ABB RobotStudio station: EstaciónDibujo_20220828-163813.rsstn

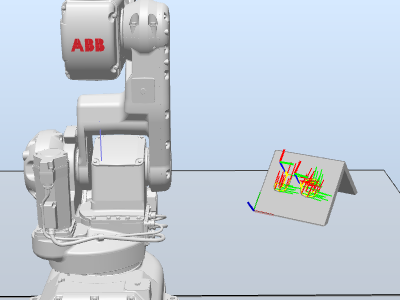
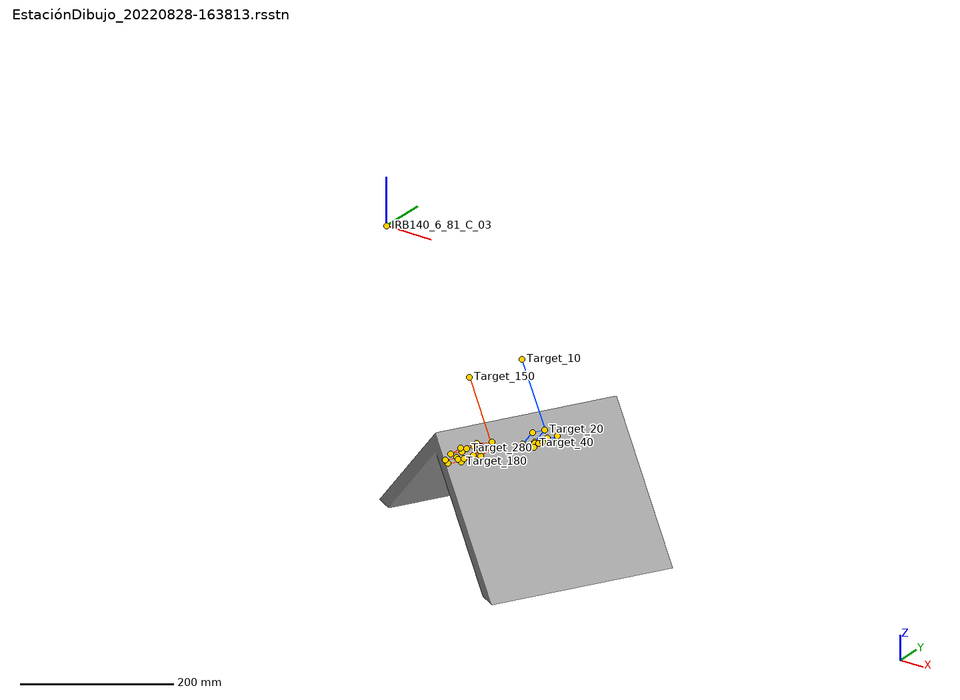
[picture v1: parts stored in the station drawn from their meshes, with robot base, taught points and paths (robot models come from the ABB library and are not in the file)]
Station EstaciónDibujo (saved by RobotStudio 22.2.9947.0)
Controller ControladorDibujo
  mechanical unit ROB_1: IRB140_6_81_C_03, 6 joints, base frame (0, 0, 0) mm
Layout (positions relative to the parent item):
  - IRB140_6_81_C_03 [mechanism, from Robots\IRB140_6_81_C_G_03.rslib] at (0, 0, 0) mm; joint values [0, 0, 0, 0, 0, 0] (rad or m)
  - Tablero [part] at (588.81, -446.49, 0) mm, rotated rx 90 ry 0 rz -120 deg, size 260 x 173.2 x 346.5 mm
  - HerramientaMarcador [mechanism] at (515, 0, 712) mm, rotated rx 0 ry 90 rz 0 deg
      TCP PuntaMarcador at (58.47, 0, 120.68) mm, rotated rx 0 ry 40 rz 0 deg
      links: HerramientaM-Marcador
  - Part_1 [part] at (588.81, -446.49, 0) mm, rotated rx 90 ry 0 rz -120 deg, size 260 x 173.2 x 173.2 mm
Attachment: HerramientaMarcador is attached to IRB140_6_81_C_03 / Link6
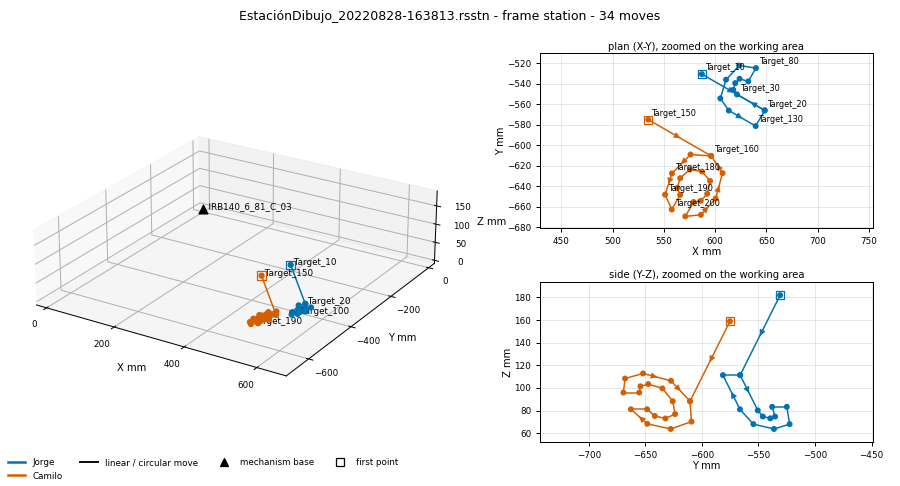
[picture p0: tool path of EstaciónDibujo_20220828-163813.rsstn in frame station, 34 of 36 moves have a stored position in this frame; points joined in program order, loops and branches not executed]
Targets, tools, work objects and paths stored in the station, written as RAPID:
! task T_ROB1
MODULE Module1
  CONST robtarget Target_10:=[[73.955465637,157.243972961,100.000985962],[-0.000003962,0.707387962,0.706825489,0.000002607],[0,0,0,0],[9E+09,9E+09,9E+09,9E+09,9E+09,9E+09]];
  CONST robtarget Target_20:=[[73.955274379,157.244902053,0.000985967],[-0.000003962,0.707387962,0.706825489,0.000002607],[0,0,0,0],[9E+09,9E+09,9E+09,9E+09,9E+09,9E+09]];
  CONST robtarget Target_30:=[[73.920195161,113.145486504,0.000576311],[-0.000003962,0.707387962,0.706825489,0.000002607],[0,0,0,0],[9E+09,9E+09,9E+09,9E+09,9E+09,9E+09]];
  CONST robtarget Target_40:=[[71.888872615,105.530963007,0.00050945],[-0.000003962,0.707387962,0.706825489,0.000002607],[0,0,0,0],[9E+09,9E+09,9E+09,9E+09,9E+09,9E+09]];
  CONST robtarget Target_50:=[[65.240745034,103.225737132,0.000500747],[-0.000003962,0.707387962,0.706825489,0.000002607],[0,0,0,0],[9E+09,9E+09,9E+09,9E+09,9E+09,9E+09]];
  CONST robtarget Target_60:=[[59.480450131,105.398209048,0.000531949],[-0.000003962,0.707387962,0.706825489,0.000002607],[0,0,0,0],[9E+09,9E+09,9E+09,9E+09,9E+09,9E+09]];
  CONST robtarget Target_70:=[[57.436372502,117.608477845,0.000649303],[-0.000003962,0.707387962,0.706825489,0.000002607],[0,0,0,0],[9E+09,9E+09,9E+09,9E+09,9E+09,9E+09]];
  CONST robtarget Target_80:=[[42.489351966,117.620367567,0.000678],[-0.000003962,0.707387962,0.706825489,0.000002607],[0,0,0,0],[9E+09,9E+09,9E+09,9E+09,9E+09,9E+09]];
  CONST robtarget Target_90:=[[48.405321169,95.993812933,0.000465755],[-0.000003962,0.707387962,0.706825489,0.000002607],[0,0,0,0],[9E+09,9E+09,9E+09,9E+09,9E+09,9E+09]];
  CONST robtarget Target_100:=[[66.827562858,89.931887143,0.0003742],[-0.000003962,0.707387962,0.706825489,0.000002607],[0,0,0,0],[9E+09,9E+09,9E+09,9E+09,9E+09,9E+09]];
  CONST robtarget Target_110:=[[85.430597019,95.992885761,0.000394933],[-0.000003962,0.707387962,0.706825489,0.000002607],[0,0,0,0],[9E+09,9E+09,9E+09,9E+09,9E+09,9E+09]];
  CONST robtarget Target_120:=[[91.549595196,114.443606918,0.000554654],[-0.000003962,0.707387962,0.706825489,0.000002607],[0,0,0,0],[9E+09,9E+09,9E+09,9E+09,9E+09,9E+09]];
  CONST robtarget Target_130:=[[91.583630659,157.230879442,0.000952121],[-0.000003962,0.707387962,0.706825489,0.000002607],[0,0,0,0],[9E+09,9E+09,9E+09,9E+09,9E+09,9E+09]];
  CONST robtarget Target_140:=[[73.955274379,157.244902053,0.000985967],[-0.000003962,0.707387962,0.706825489,0.000002607],[0,0,0,0],[9E+09,9E+09,9E+09,9E+09,9E+09,9E+09]];
  CONST jointtarget Home:=[[0,0,0,0,0,0],[9E+09,9E+09,9E+09,9E+09,9E+09,9E+09]];
  CONST robtarget Target_150:=[[138.452714894,124.560220972,100.000558944],[0.000004101,0.745570763,0.666426468,0.000002383],[0,0,0,0],[9E+09,9E+09,9E+09,9E+09,9E+09,9E+09]];
  CONST robtarget Target_160:=[[138.452523635,124.561150062,0.000558949],[0.000004101,0.745570763,0.666426468,0.000002383],[0,0,0,0],[9E+09,9E+09,9E+09,9E+09,9E+09,9E+09]];
  CONST robtarget Target_170:=[[147.331968493,99.024331413,0.000304705],[0.000004101,0.745570763,0.666426468,0.000002383],[0,0,0,0],[9E+09,9E+09,9E+09,9E+09,9E+09,9E+09]];
  CONST robtarget Target_180:=[[172.255402363,89.848023763,0.00017178],[0.000004101,0.745570763,0.666426468,0.000002383],[0,0,0,0],[9E+09,9E+09,9E+09,9E+09,9E+09,9E+09]];
  CONST robtarget Target_190:=[[193.568592092,96.27768983,0.000190755],[0.000004101,0.745570763,0.666426468,0.000002383],[0,0,0,0],[9E+09,9E+09,9E+09,9E+09,9E+09,9E+09]];
  CONST robtarget Target_200:=[[202.91069392,114.469123347,0.000341902],[0.000004101,0.745570763,0.666426468,0.000002383],[0,0,0,0],[9E+09,9E+09,9E+09,9E+09,9E+09,9E+09]];
  CONST robtarget Target_210:=[[186.423331573,114.482238345,0.000373558],[0.000004101,0.745570763,0.666426468,0.000002383],[0,0,0,0],[9E+09,9E+09,9E+09,9E+09,9E+09,9E+09]];
  CONST robtarget Target_220:=[[181.881209734,106.099540689,0.000304363],[0.000004101,0.745570763,0.666426468,0.000002383],[0,0,0,0],[9E+09,9E+09,9E+09,9E+09,9E+09,9E+09]];
  CONST robtarget Target_230:=[[172.322889602,102.969408624,0.000293562],[0.000004101,0.745570763,0.666426468,0.000002383],[0,0,0,0],[9E+09,9E+09,9E+09,9E+09,9E+09,9E+09]];
  CONST robtarget Target_240:=[[160.26125798,108.484302356,0.000367869],[0.000004101,0.745570763,0.666426468,0.000002383],[0,0,0,0],[9E+09,9E+09,9E+09,9E+09,9E+09,9E+09]];
  CONST robtarget Target_250:=[[156.080834535,124.490077756,0.000524572],[0.000004101,0.745570763,0.666426468,0.000002383],[0,0,0,0],[9E+09,9E+09,9E+09,9E+09,9E+09,9E+09]];
  CONST robtarget Target_260:=[[160.144183026,140.60339505,0.000666508],[0.000004101,0.745570763,0.666426468,0.000002383],[0,0,0,0],[9E+09,9E+09,9E+09,9E+09,9E+09,9E+09]];
  CONST robtarget Target_270:=[[172.357106589,145.984879936,0.000693148],[0.000004673,-0.031268643,0.999511016,0.000000809],[0,0,0,0],[9E+09,9E+09,9E+09,9E+09,9E+09,9E+09]];
  CONST robtarget Target_280:=[[181.48283441,143.182183899,0.000649655],[0.000004673,-0.031268643,0.999511016,0.000000809],[0,0,0,0],[9E+09,9E+09,9E+09,9E+09,9E+09,9E+09]];
  CONST robtarget Target_290:=[[185.926493609,135.362835763,0.000568508],[0.000004585,0.055963469,0.998432817,0.000001213],[0,0,0,0],[9E+09,9E+09,9E+09,9E+09,9E+09,9E+09]];
  CONST robtarget Target_300:=[[202.071557775,135.349993048,0.00053751],[0.000004673,-0.031268643,0.999511016,0.000000809],[0,0,0,0],[9E+09,9E+09,9E+09,9E+09,9E+09,9E+09]];
  CONST robtarget Target_310:=[[193.214284478,152.899831469,0.000717503],[0.000004673,-0.031268643,0.999511016,0.000000809],[0,0,0,0],[9E+09,9E+09,9E+09,9E+09,9E+09,9E+09]];
  CONST robtarget Target_320:=[[172.253580878,159.277550028,0.000816848],[0.000004673,-0.031268643,0.999511016,0.000000809],[0,0,0,0],[9E+09,9E+09,9E+09,9E+09,9E+09,9E+09]];
  CONST robtarget Target_330:=[[147.429633844,150.083764579,0.000778907],[0.000004101,0.745570763,0.666426468,0.000002383],[0,0,0,0],[9E+09,9E+09,9E+09,9E+09,9E+09,9E+09]];
  CONST robtarget Target_340:=[[138.452523635,124.561150062,0.000558949],[0.000004101,0.745570763,0.666426468,0.000002383],[0,0,0,0],[9E+09,9E+09,9E+09,9E+09,9E+09,9E+09]];
  CONST jointtarget Cerca:=[[0,30,3,0,30,0],[9E+09,9E+09,9E+09,9E+09,9E+09,9E+09]];
  PROC main()
  ENDPROC
  PROC Jorge()
    MoveL Target_10,v200,z10,PuntaMarcador\WObj:=SuperficieTablero;
    MoveL Target_20,v200,z10,PuntaMarcador\WObj:=SuperficieTablero;
    MoveL Target_30,v200,z10,PuntaMarcador\WObj:=SuperficieTablero;
    MoveL Target_40,v200,z10,PuntaMarcador\WObj:=SuperficieTablero;
    MoveL Target_50,v200,z10,PuntaMarcador\WObj:=SuperficieTablero;
    MoveL Target_60,v200,z10,PuntaMarcador\WObj:=SuperficieTablero;
    MoveL Target_70,v200,z10,PuntaMarcador\WObj:=SuperficieTablero;
    MoveL Target_80,v200,z10,PuntaMarcador\WObj:=SuperficieTablero;
    MoveL Target_90,v200,z10,PuntaMarcador\WObj:=SuperficieTablero;
    MoveL Target_100,v200,z10,PuntaMarcador\WObj:=SuperficieTablero;
    MoveL Target_110,v200,z10,PuntaMarcador\WObj:=SuperficieTablero;
    MoveL Target_120,v200,z10,PuntaMarcador\WObj:=SuperficieTablero;
    MoveL Target_130,v200,z10,PuntaMarcador\WObj:=SuperficieTablero;
    MoveL Target_140,v200,z10,PuntaMarcador\WObj:=SuperficieTablero;
  ENDPROC
  PROC Camilo()
    MoveL Target_150,v200,z10,PuntaMarcador\WObj:=SuperficieTablero;
    MoveL Target_160,v200,z10,PuntaMarcador\WObj:=SuperficieTablero;
    MoveL Target_170,v200,z10,PuntaMarcador\WObj:=SuperficieTablero;
    MoveL Target_180,v200,z10,PuntaMarcador\WObj:=SuperficieTablero;
    MoveL Target_190,v200,z10,PuntaMarcador\WObj:=SuperficieTablero;
    MoveL Target_200,v200,z10,PuntaMarcador\WObj:=SuperficieTablero;
    MoveL Target_210,v200,z10,PuntaMarcador\WObj:=SuperficieTablero;
    MoveL Target_220,v200,z10,PuntaMarcador\WObj:=SuperficieTablero;
    MoveL Target_230,v200,z10,PuntaMarcador\WObj:=SuperficieTablero;
    MoveL Target_240,v200,z10,PuntaMarcador\WObj:=SuperficieTablero;
    MoveL Target_250,v200,z10,PuntaMarcador\WObj:=SuperficieTablero;
    MoveL Target_260,v200,z10,PuntaMarcador\WObj:=SuperficieTablero;
    MoveL Target_270,v200,z10,PuntaMarcador\WObj:=SuperficieTablero;
    MoveL Target_280,v200,z10,PuntaMarcador\WObj:=SuperficieTablero;
    MoveL Target_290,v200,z10,PuntaMarcador\WObj:=SuperficieTablero;
    MoveL Target_300,v200,z10,PuntaMarcador\WObj:=SuperficieTablero;
    MoveL Target_310,v200,z10,PuntaMarcador\WObj:=SuperficieTablero;
    MoveL Target_320,v200,z10,PuntaMarcador\WObj:=SuperficieTablero;
    MoveL Target_330,v200,z10,PuntaMarcador\WObj:=SuperficieTablero;
    MoveL Target_340,v200,z10,PuntaMarcador\WObj:=SuperficieTablero;
  ENDPROC
  PROC AHome()
    MoveAbsJ Home,v200,z10,PuntaMarcador\WObj:=SuperficieTablero;
  ENDPROC
  PROC Acerca()
    MoveAbsJ Cerca,v200,z10,PuntaMarcador\WObj:=SuperficieTablero;
  ENDPROC
ENDMODULE

! task T_ROB1
MODULE CalibData
  PERS tooldata PuntaMarcador:=[TRUE,[[58.468,0,120.677],[0.939692621,0,0.342020143,0]],[1,[6.317,0,37.933],[1,0,0,0],0,0,0]];
  TASK PERS wobjdata SuperficieTablero:=[FALSE,TRUE,"",[[0,0,0],[1,0,0,0]],[[588.848204459,-446.615736766,0.09457014],[0.462258525,0.191206976,-0.331486376,-0.799921078]]];
ENDMODULE

